Staubli VAL3: fhmns.pgx

public program fhmns(num x_nSec, string& x_sHMinSec[])
  local num l_nHour
  local num l_nMin
  local num l_nSec
begin
  //-----------------------------------------------------------------------
  //Header begin
  //Description of program
  //  Convert a num seconds in string hour : "xx h xx mn xx s".
  //
  //Input parameters
  //  num x_nSec :
  //    role : put a numerical expression that you want to convert in Hmns
  //
  //Output parameters
  //  string x_sHMinSec :
  //    role : string hour correspond of your numerical expression
  //
  //Example
  //  call hmns(l_nSecond,l_sHMinSec)
  //
  //History
  //  Creation : 28-04-08 - f.Rob
  //Header end
  //-----------------------------------------------------------------------
  l_nHour=roundDown(x_nSec/3600)
  l_nMin=roundDown((x_nSec%3600)/60)
  l_nSec=roundDown(x_nSec-l_nHour*3600-l_nMin*60)
  x_sHMinSec=toString("3.0",l_nHour)+" h "+toString("2.0",l_nMin)+" mn "+toString("2.0",l_nSec)+" s"
end
